FUNCTION WRITE_ANY_UDINT : BOOL
VAR_INPUT
    ptr: POINTER TO UDINT;
    val: UDINT;
END_VAR

ptr^ := val;

END_FUNCTION

(* stored: Version 1.1.0.1, ProductVersion 3.1.4022.9
   POU WRITE_ANY_UDINT: Id {268b342f-fd80-4091-8fb8-f5f8dab7958d}, SpecialFunc None *)
